FUNCTION_BLOCK fbMotorDirectCtrl

VAR_INPUT
	IN_DevName:STRING;
	In_Enable:BOOL;
	In_Reset:BOOL;

	(*Starter Healthy Signal*)
	In_StarterOK:BOOL;

END_VAR

VAR_OUTPUT
	Out_MotorOn:BOOL;

END_VAR

VAR_IN_OUT
	MotorVar:structMotorDirect;	
	Station:structStationCtrl;
END_VAR


VAR

	MotorOn:BOOL;
	On_TOut: TON;
	On_TON: TON;
	Loc_OnPls: BOOL;
	OnPls: R_TRIG;
	Out_RSErr:BOOL;
	OnPosPls: F_TRIG;

	pls_ManualModeOff: R_TRIG;
END_VAR

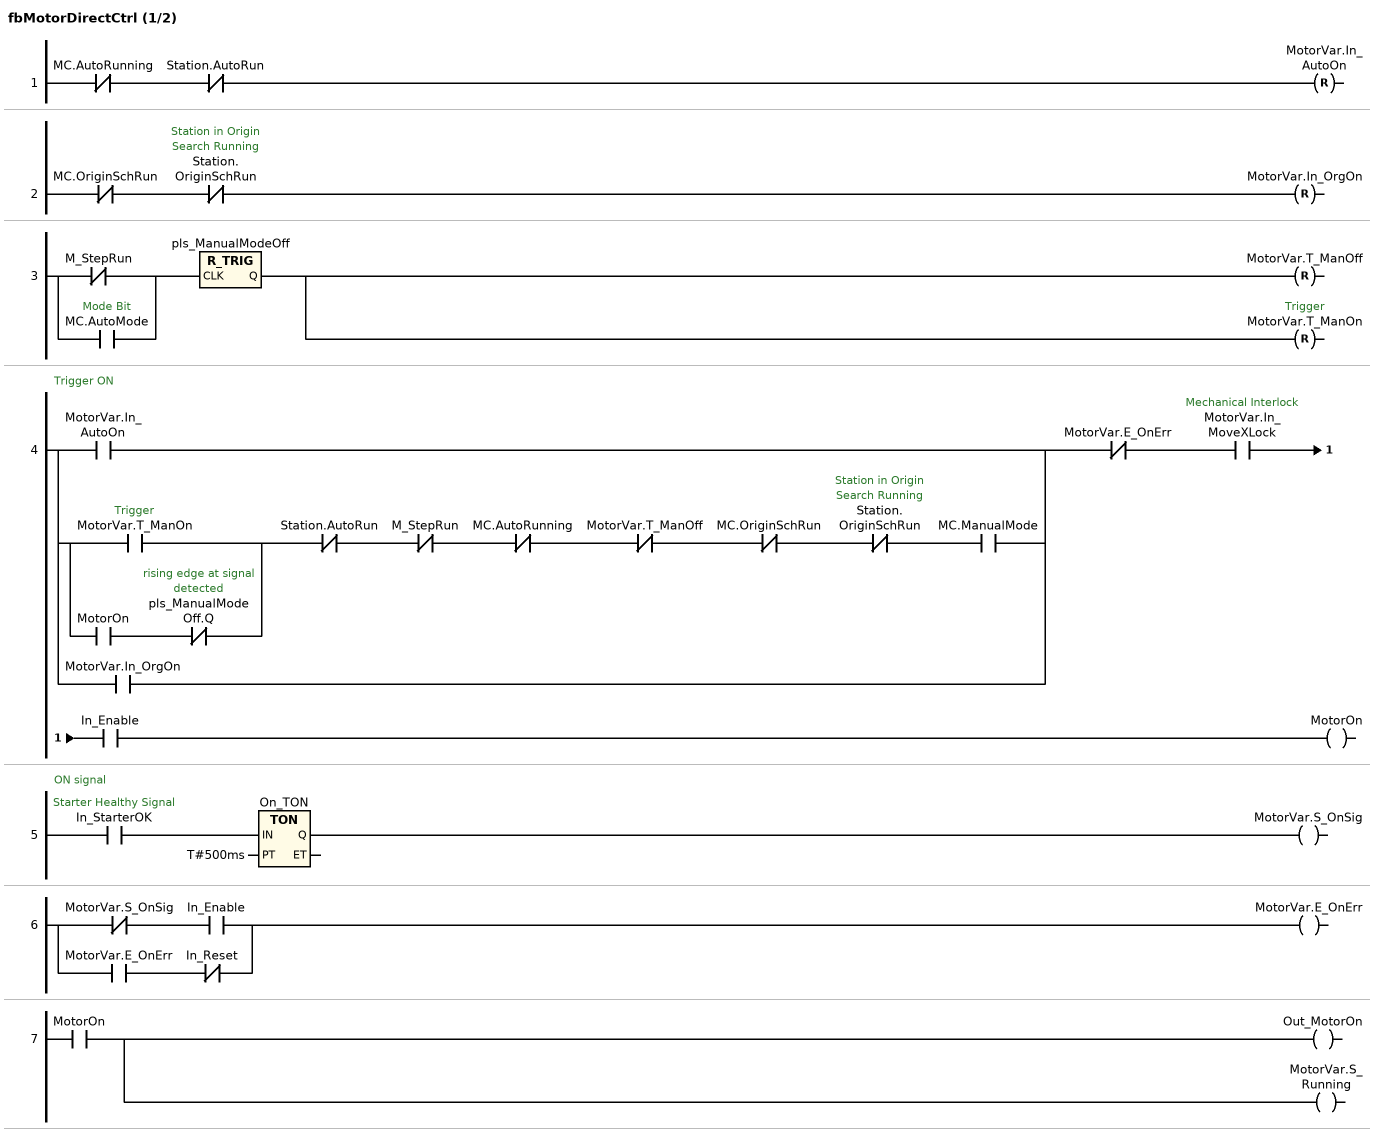
// NETWORK 1
MotorVar.In_AutoOn R= NOT MC.AutoRunning AND NOT Station.AutoRun;

// NETWORK 2
//   Station.OriginSchRun: Station in Origin Search Running
MotorVar.In_OrgOn R= NOT MC.OriginSchRun AND NOT Station.OriginSchRun;

// NETWORK 3
//   MC.AutoMode: Mode Bit
//   MotorVar.T_ManOn: Trigger
pls_ManualModeOff(CLK := NOT M_StepRun OR MC.AutoMode); // R_TRIG
MotorVar.T_ManOff R= pls_ManualModeOff.Q;
MotorVar.T_ManOn R= pls_ManualModeOff.Q;

// NETWORK 4
// Trigger ON
//   MotorVar.T_ManOn: Trigger
//   pls_ManualModeOff.Q: rising edge at signal detected
//   Station.OriginSchRun: Station in Origin Search Running
//   MotorVar.In_MoveXLock: Mechanical Interlock
MotorOn := (MotorVar.In_AutoOn OR (MotorVar.T_ManOn OR MotorOn AND NOT pls_ManualModeOff.Q) AND NOT Station.AutoRun AND NOT M_StepRun AND NOT MC.AutoRunning AND NOT MotorVar.T_ManOff AND NOT MC.OriginSchRun AND NOT Station.OriginSchRun AND MC.ManualMode OR MotorVar.In_OrgOn) AND NOT MotorVar.E_OnErr AND MotorVar.In_MoveXLock AND In_Enable;

// NETWORK 5
// ON signal
//   In_StarterOK: Starter Healthy Signal
On_TON(IN := In_StarterOK, PT := T#500ms); // TON
MotorVar.S_OnSig := On_TON.Q;

// NETWORK 6
MotorVar.E_OnErr := NOT MotorVar.S_OnSig AND In_Enable OR MotorVar.E_OnErr AND NOT In_Reset;

// NETWORK 7
Out_MotorOn := MotorOn;
MotorVar.S_Running := MotorOn;

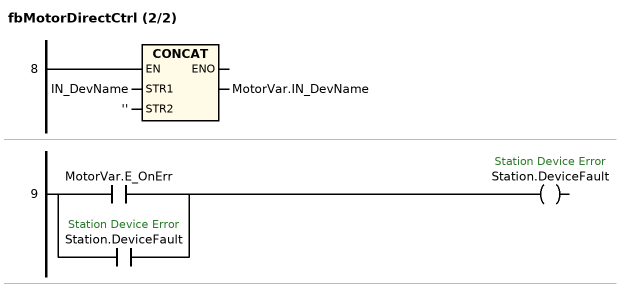
// NETWORK 8
MotorVar.IN_DevName := CONCAT(STR1 := IN_DevName, STR2 := '');

// NETWORK 9
//   Station.DeviceFault: Station Device Error
Station.DeviceFault := MotorVar.E_OnErr OR Station.DeviceFault;

END_FUNCTION_BLOCK

(* stored: Version 1.1.0.1, ProductVersion 3.1.4018.2
   POU fbMotorDirectCtrl: Id {6cf8fa1c-3ce9-4b6c-82aa-9a2ab1d38e7e}, SpecialFunc None *)
